% RSLogix 500 project LVD190506v3_Bot.RSS, saved by version 11.00.00.00 %
PROJECT "LINCEBOT"    % processor: MicroLogix 1400 %

PROGRAM FILES
  LAD 2 "MAIN"  40 rungs  % Main Program Routine %
  LAD 4 "PACKAGER"  27 rungs  % normal %
  LAD 5 "NO PACKAGE"  7 rungs
  LAD 6 "TIMING"  11 rungs  % normal %
  LAD 8 "LOOP TIME"  6 rungs
  LAD 10 "AIR PRESUR"  2 rungs
  LAD 12 "ENABLES"  13 rungs
  LAD 14 "SPEED OUT"  10 rungs
  LAD 16 "TOTALCOUNT"  4 rungs
  LAD 18 "TESTTRIG1"  4 rungs
  LAD 24 "SKIPPED"  5 rungs
  LAD 70 "ALIGNFAILS"  4 rungs  % normal %
  LAD 80 "HSC BOT"  5 rungs
  LAD 100 "1 MS STI"  19 rungs  % high speed %
  LAD 102 "SPEED BOT"  8 rungs  % high speed %
  LAD 104 "P BOT"  9 rungs  % high speed %
  LAD 110 "SHIFT BOT"  10 rungs
  LAD 120 "BOTOPTIC"  3 rungs
  LAD 121 "BOTOPTMES"  8 rungs
  LAD 129   1 rungs  % used for analysis %
  LAD 130 "INS1"  21 rungs
  LAD 131 "INS1RESULT"  7 rungs
  LAD 132 "INS1PASS"  3 rungs
  LAD 133 "INS1FAIL"  3 rungs
  LAD 134 "INS1ACQ"  8 rungs
  LAD 135 "Q1TIMETEST"  5 rungs
  LAD 136 "INS1TRIG"  5 rungs
  LAD 137 "FIFO1SET"  9 rungs
  LAD 138 "FIFO1GET"  8 rungs
  LAD 139 "INSDATA1"  3 rungs  % used for analysis %
  LAD 140 "TESTFAULT1"  9 rungs
  LAD 141 "INS1FIX1"  6 rungs
  LAD 142 "INS1FIX2"  3 rungs
  LAD 143 "HS TRIG1"  5 rungs
  LAD 200 "XFEROUT"  3 rungs
  LAD 201 "XFER GOOD"  5 rungs
  LAD 202 "XFER NG"  5 rungs
  LAD 222 "RATE1"  9 rungs
  LAD 223 "RATE2"  6 rungs
  LAD 224 "RESET RATE"  6 rungs
  LAD 122, 123, 124, 125, 126, 127, 128, 144, 145: only END

DATA FILES
  O0 OUTPUT  11 elements
  I1 INPUT  11 elements
  S2 STATUS  66 elements
  B3 BINARY  14 elements
  T4 TIMER  40 elements
  C5 COUNTER  1 elements
  R6 CONTROL  20 elements
  N7 INTEGER  200 elements
  F8 FLOAT  100 elements
  B9 TOP BS DAT  256 elements
  B10 OLD_COM  1 elements
  B11 BOT BS DAT  256 elements
  B12 HMI_BINARY  22 elements  % general use with hmi to avoid additional reads %
  L13  COUNTS  256 elements
  F14 HMI_FLOATS  100 elements
  N15 HMI_INTS  100 elements
  L16 HMI_LONGS  100 elements
  B17 SIDE DATA  128 elements
  B18 TOP DATA  128 elements
  L19 INS1TIME  10 elements
  L20 INS1POS  10 elements
  L21 INS5TIME  10 elements
  L22 INS5POS  10 elements
  L23 NEW READ  100 elements
  L24 NEW WRITE  100 elements
  L25 INS6TIME  10 elements
  L26 INS6POS  10 elements
  L27 RATETIMES  50 elements
  L28 INS1TIME  50 elements
  L29 INS1POS  50 elements
  L42   52 elements
  B181 BLANK  256 elements  % used to wipe bs files %
  F182 TEST FLOAT  50 elements
  L183 TEST LONG  50 elements
  N184 TEST INTS  50 elements
  B185 TEST BITS  50 elements
  N186 HMI INTS  50 elements
  L187 HMI LONG  50 elements
  F188 HMI FLOAT  50 elements
  B189 HMI BITS  50 elements
  L190 COUNTS  50 elements
  B191 ERROR BITS  10 elements
  L192 SPD OFFSET  50 elements
  F193 SPD OFFSET  50 elements
  B194 BOT GOOD  128 elements
  B195 BOT NG  128 elements
  B196 CTRL BITS  50 elements
  N197 CTRL INTS  50 elements
  B198 TRK BITS  50 elements
  L199 TRK LONG  50 elements
  N200 TRK INTS  50 elements
  L201 INS LONG  50 elements
  B202 INS BITS  50 elements
  N203 INS INTS  50 elements
  L204 CTRL LONG  50 elements
  F205 CTRL FLTS  50 elements

LADDER 2 "MAIN"    % Main Program Routine %
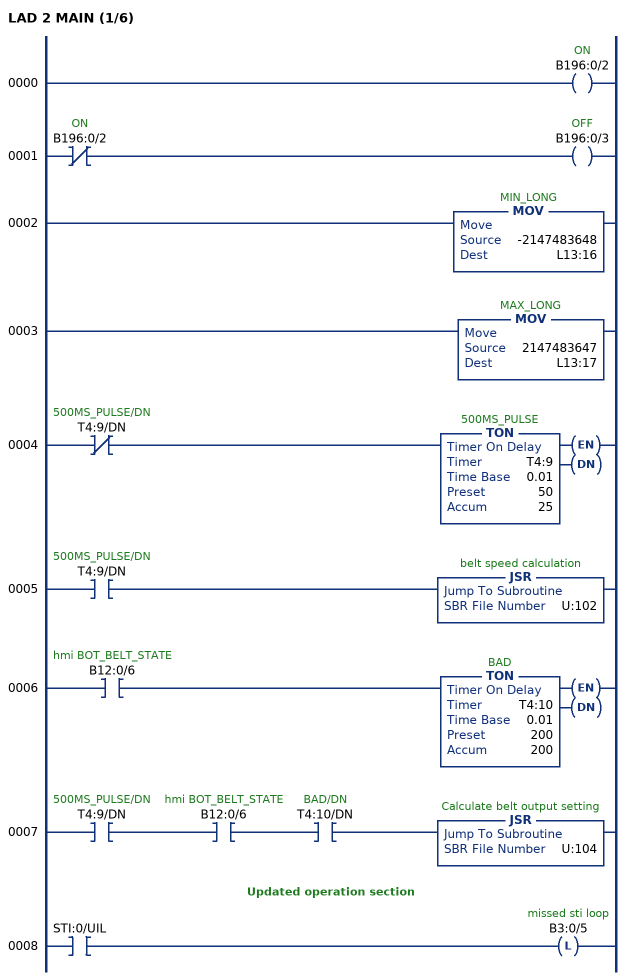
% Rung: 0 %
SOR OTE B196:0/2 EOR
%   B196:0/2  ON %
% Rung: 1 %
SOR XIO B196:0/2 OTE B196:0/3 EOR
%   B196:0/2  ON %
%   B196:0/3  OFF %
% Rung: 2 %
SOR MOV -2147483648 L13:16 EOR
%   L13:16  MIN_LONG %
% Rung: 3 %
SOR MOV 2147483647 L13:17 EOR
%   L13:17  MAX_LONG %
% Rung: 4 %
SOR XIO T4:9/DN TON T4:9 0.01 50 25 EOR
%   T4:9  500MS_PULSE %
% Rung: 5 %
SOR XIC T4:9/DN JSR U:102 EOR
%   T4:9  500MS_PULSE %
%   U:102  "belt speed calculation" %
% Rung: 6 %
SOR XIC B12:0/6 TON T4:10 0.01 200 200 EOR
%   B12:0/6  BOT_BELT_STATE  "hmi" %
%   T4:10  BAD %
% Rung: 7 %
SOR XIC T4:9/DN XIC B12:0/6 XIC T4:10/DN JSR U:104 EOR
%   T4:9  500MS_PULSE %
%   B12:0/6  BOT_BELT_STATE  "hmi" %
%   T4:10  BAD %
%   U:104  "Calculate belt output setting" %
% Rung: 8 %
% TITLE: Updated operation section %
SOR XIC STI:0/UIL OTL B3:0/5 EOR
%   B3:0/5  "missed sti loop" %

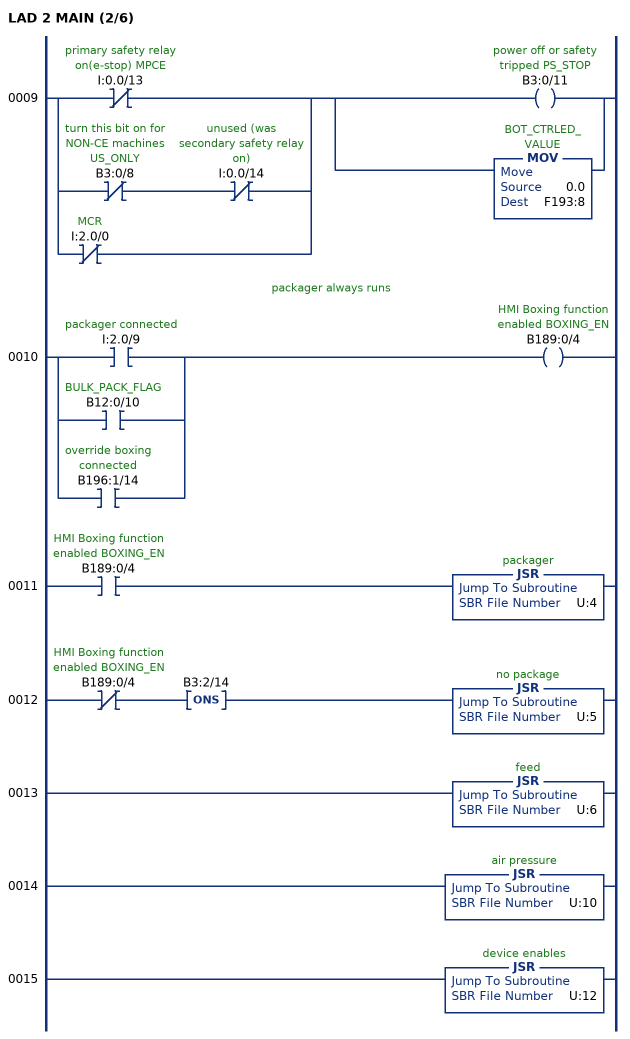
% Rung: 9 %
SOR BST XIO I:0.0/13 NXB XIO B3:0/8 XIO I:0.0/14 NXB XIO I:2.0/0 BND BST OTE B3:0/11 NXB MOV 0.0 F193:8 BND EOR
%   I:0.0/13  MPCE  "primary safety relay on(e-stop)" %
%   B3:0/8  US_ONLY  "turn this bit on for NON-CE machines" %
%   I:0.0/14  "unused (was secondary safety relay on)" %
%   I:2.0/0  MCR %
%   B3:0/11  PS_STOP  "power off or safety tripped" %
%   F193:8  BOT_CTRLED_VALUE %
% Rung: 10 %
% packager always runs %
SOR BST XIC I:2.0/9 NXB XIC B12:0/10 NXB XIC B196:1/14 BND OTE B189:0/4 EOR
%   I:2.0/9  "packager connected" %
%   B12:0/10  BULK_PACK_FLAG %
%   B196:1/14  "override boxing connected" %
%   B189:0/4  BOXING_EN  "HMI Boxing function enabled" %
% Rung: 11 %
SOR XIC B189:0/4 JSR U:4 EOR
%   B189:0/4  BOXING_EN  "HMI Boxing function enabled" %
%   U:4  "packager" %
% Rung: 12 %
SOR XIO B189:0/4 ONS B3:2/14 JSR U:5 EOR
%   B189:0/4  BOXING_EN  "HMI Boxing function enabled" %
%   U:5  "no package" %
% Rung: 13 %
SOR JSR U:6 EOR
%   U:6  "feed" %
% Rung: 14 %
SOR JSR U:10 EOR
%   U:10  "air pressure" %
% Rung: 15 %
SOR JSR U:12 EOR
%   U:12  "device enables" %

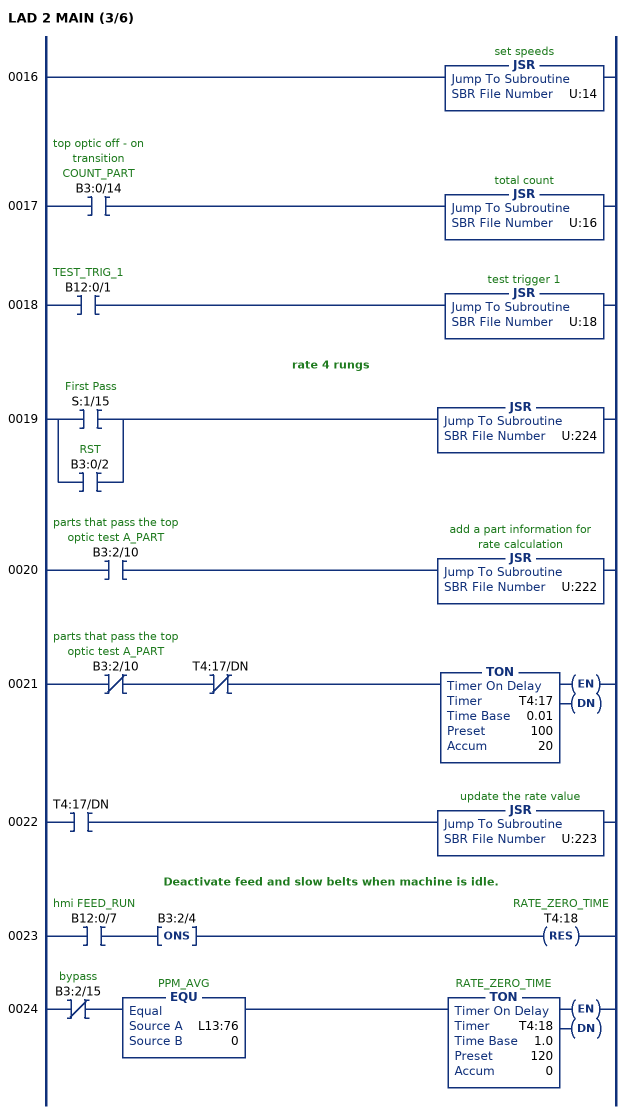
% Rung: 16 %
SOR JSR U:14 EOR
%   U:14  "set speeds" %
% Rung: 17 %
SOR XIC B3:0/14 JSR U:16 EOR
%   B3:0/14  COUNT_PART  "top optic off - on transition" %
%   U:16  "total count" %
% Rung: 18 %
SOR XIC B12:0/1 JSR U:18 EOR
%   B12:0/1  TEST_TRIG_1 %
%   U:18  "test trigger 1" %
% Rung: 19 %
% TITLE: rate 4 rungs %
SOR BST XIC S:1/15 NXB XIC B3:0/2 BND JSR U:224 EOR
%   S:1/15  "First Pass" %
%   B3:0/2  RST %
% Rung: 20 %
SOR XIC B3:2/10 JSR U:222 EOR
%   B3:2/10  A_PART  "parts that pass the top optic test" %
%   U:222  "add a part information for rate calculation" %
% Rung: 21 %
SOR XIO B3:2/10 XIO T4:17/DN TON T4:17 0.01 100 20 EOR
%   B3:2/10  A_PART  "parts that pass the top optic test" %
% Rung: 22 %
SOR XIC T4:17/DN JSR U:223 EOR
%   U:223  "update the rate value" %
% Rung: 23 %
% TITLE: Deactivate feed and slow belts when machine is idle. %
SOR XIC B12:0/7 ONS B3:2/4 RES T4:18 EOR
%   B12:0/7  FEED_RUN  "hmi" %
%   T4:18  RATE_ZERO_TIME %
% Rung: 24 %
SOR XIO B3:2/15 EQU L13:76 0 TON T4:18 1.0 120 0 EOR
%   B3:2/15  "bypass" %
%   L13:76  PPM_AVG %
%   T4:18  RATE_ZERO_TIME %

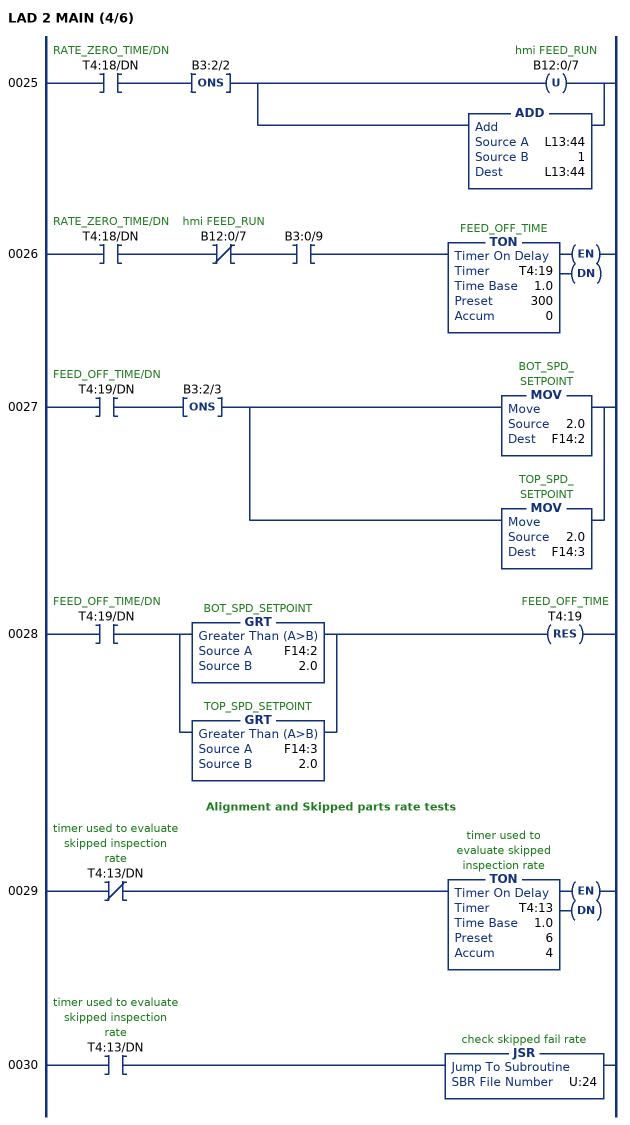
% Rung: 25 %
SOR XIC T4:18/DN ONS B3:2/2 BST OTU B12:0/7 NXB ADD L13:44 1 L13:44 BND EOR
%   T4:18  RATE_ZERO_TIME %
%   B12:0/7  FEED_RUN  "hmi" %
% Rung: 26 %
SOR XIC T4:18/DN XIO B12:0/7 XIC B3:0/9 TON T4:19 1.0 300 0 EOR
%   T4:18  RATE_ZERO_TIME %
%   B12:0/7  FEED_RUN  "hmi" %
%   T4:19  FEED_OFF_TIME %
% Rung: 27 %
SOR XIC T4:19/DN ONS B3:2/3 BST MOV 2.0 F14:2 NXB MOV 2.0 F14:3 BND EOR
%   T4:19  FEED_OFF_TIME %
%   F14:2  BOT_SPD_SETPOINT %
%   F14:3  TOP_SPD_SETPOINT %
% Rung: 28 %
SOR XIC T4:19/DN BST GRT F14:2 2.0 NXB GRT F14:3 2.0 BND RES T4:19 EOR
%   T4:19  FEED_OFF_TIME %
%   F14:2  BOT_SPD_SETPOINT %
%   F14:3  TOP_SPD_SETPOINT %
% Rung: 29 %
% TITLE: Alignment and Skipped parts rate tests %
SOR XIO T4:13/DN TON T4:13 1.0 6 4 EOR
%   T4:13  "timer used to evaluate skipped inspection rate" %
% Rung: 30 %
SOR XIC T4:13/DN JSR U:24 EOR
%   T4:13  "timer used to evaluate skipped inspection rate" %
%   U:24  "check skipped fail rate" %

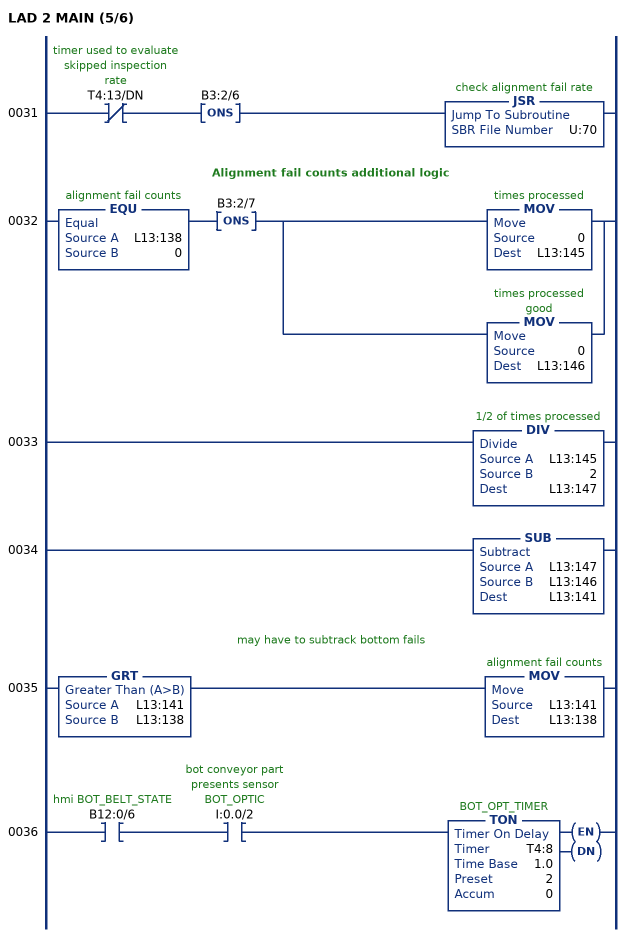
% Rung: 31 %
SOR XIO T4:13/DN ONS B3:2/6 JSR U:70 EOR
%   T4:13  "timer used to evaluate skipped inspection rate" %
%   U:70  "check alignment fail rate" %
% Rung: 32 %
% TITLE: Alignment fail counts additional logic %
SOR EQU L13:138 0 ONS B3:2/7 BST MOV 0 L13:145 NXB MOV 0 L13:146 BND EOR
%   L13:138  "alignment fail counts" %
%   L13:145  "times processed" %
%   L13:146  "times processed good" %
% Rung: 33 %
SOR DIV L13:145 2 L13:147 EOR
%   L13:145  "times processed" %
%   L13:147  "1/2 of times processed" %
% Rung: 34 %
SOR SUB L13:147 L13:146 L13:141 EOR
%   L13:147  "1/2 of times processed" %
%   L13:146  "times processed good" %
% Rung: 35 %
% may have to subtrack bottom fails %
SOR GRT L13:141 L13:138 MOV L13:141 L13:138 EOR
%   L13:138  "alignment fail counts" %
% Rung: 36 %
SOR XIC B12:0/6 XIC I:0.0/2 TON T4:8 1.0 2 0 EOR
%   B12:0/6  BOT_BELT_STATE  "hmi" %
%   I:0.0/2  BOT_OPTIC  "bot conveyor part presents sensor" %
%   T4:8  BOT_OPT_TIMER %

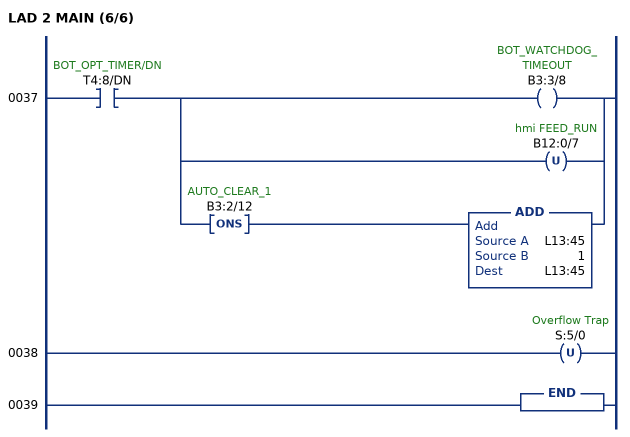
% Rung: 37 %
SOR XIC T4:8/DN BST OTE B3:3/8 NXB OTU B12:0/7 NXB ONS B3:2/12 ADD L13:45 1 L13:45 BND EOR
%   T4:8  BOT_OPT_TIMER %
%   B3:3/8  BOT_WATCHDOG_TIMEOUT %
%   B12:0/7  FEED_RUN  "hmi" %
%   B3:2/12  AUTO_CLEAR_1 %
% Rung: 38 %
SOR OTU S:5/0 EOR
%   S:5/0  "Overflow Trap" %
% Rung: 39 %
SOR END EOR

LADDER 4 "PACKAGER"    % normal %
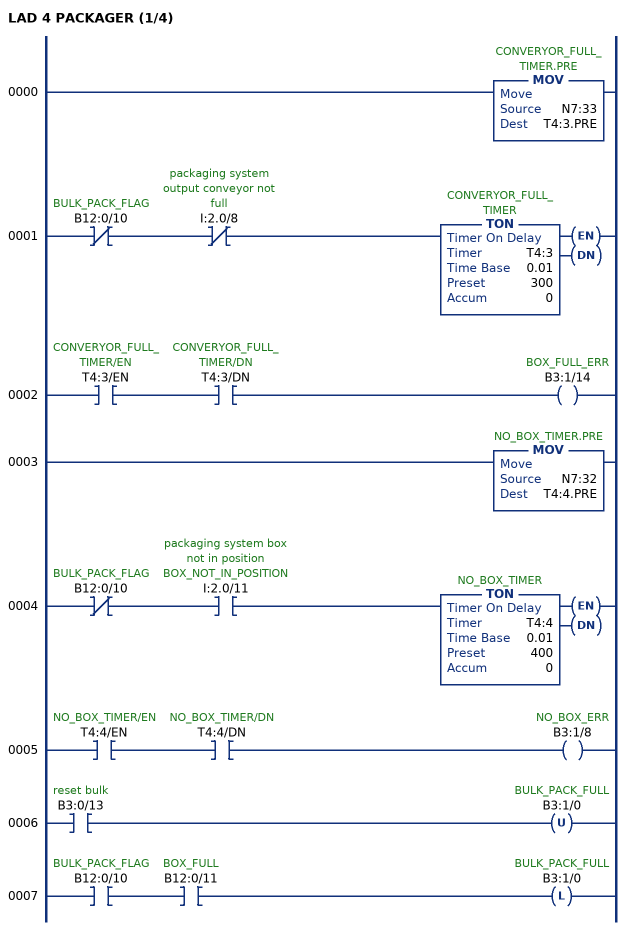
% Rung: 0 %
SOR MOV N7:33 T4:3.PRE EOR
%   T4:3  CONVERYOR_FULL_TIMER %
% Rung: 1 %
SOR XIO B12:0/10 XIO I:2.0/8 TON T4:3 0.01 300 0 EOR
%   B12:0/10  BULK_PACK_FLAG %
%   I:2.0/8  "packaging system output conveyor not full" %
%   T4:3  CONVERYOR_FULL_TIMER %
% Rung: 2 %
SOR XIC T4:3/EN XIC T4:3/DN OTE B3:1/14 EOR
%   T4:3  CONVERYOR_FULL_TIMER %
%   B3:1/14  BOX_FULL_ERR %
% Rung: 3 %
SOR MOV N7:32 T4:4.PRE EOR
%   T4:4  NO_BOX_TIMER %
% Rung: 4 %
SOR XIO B12:0/10 XIC I:2.0/11 TON T4:4 0.01 400 0 EOR
%   B12:0/10  BULK_PACK_FLAG %
%   I:2.0/11  BOX_NOT_IN_POSITION  "packaging system box not in position" %
%   T4:4  NO_BOX_TIMER %
% Rung: 5 %
SOR XIC T4:4/EN XIC T4:4/DN OTE B3:1/8 EOR
%   T4:4  NO_BOX_TIMER %
%   B3:1/8  NO_BOX_ERR %
% Rung: 6 %
SOR XIC B3:0/13 OTU B3:1/0 EOR
%   B3:0/13  "reset bulk" %
%   B3:1/0  BULK_PACK_FULL %
% Rung: 7 %
SOR XIC B12:0/10 XIC B12:0/11 OTL B3:1/0 EOR
%   B12:0/10  BULK_PACK_FLAG %
%   B12:0/11  BOX_FULL %
%   B3:1/0  BULK_PACK_FULL %

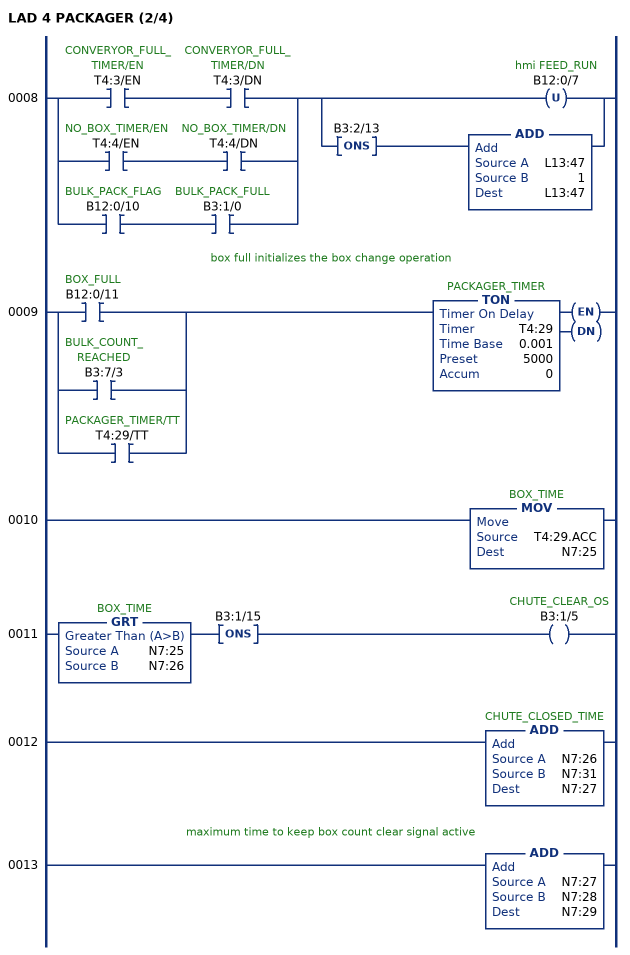
% Rung: 8 %
SOR BST XIC T4:3/EN XIC T4:3/DN NXB XIC T4:4/EN XIC T4:4/DN NXB XIC B12:0/10 XIC B3:1/0 BND BST OTU B12:0/7 NXB ONS B3:2/13 ADD L13:47 1 L13:47 BND EOR
%   T4:3  CONVERYOR_FULL_TIMER %
%   T4:4  NO_BOX_TIMER %
%   B12:0/10  BULK_PACK_FLAG %
%   B3:1/0  BULK_PACK_FULL %
%   B12:0/7  FEED_RUN  "hmi" %
% Rung: 9 %
% box full initializes the box change operation %
SOR BST XIC B12:0/11 NXB XIC B3:7/3 NXB XIC T4:29/TT BND TON T4:29 0.001 5000 0 EOR
%   B12:0/11  BOX_FULL %
%   B3:7/3  BULK_COUNT_REACHED %
%   T4:29  PACKAGER_TIMER %
% Rung: 10 %
SOR MOV T4:29.ACC N7:25 EOR
%   T4:29  PACKAGER_TIMER %
%   N7:25  BOX_TIME %
% Rung: 11 %
SOR GRT N7:25 N7:26 ONS B3:1/15 OTE B3:1/5 EOR
%   N7:25  BOX_TIME %
%   N7:26  CHUTE_CLEAR_TIME %
%   B3:1/5  CHUTE_CLEAR_OS %
% Rung: 12 %
SOR ADD N7:26 N7:31 N7:27 EOR
%   N7:26  CHUTE_CLEAR_TIME %
%   N7:27  CHUTE_CLOSED_TIME %
% Rung: 13 %
% maximum time to keep box count clear signal active %
SOR ADD N7:27 N7:28 N7:29 EOR
%   N7:27  CHUTE_CLOSED_TIME %

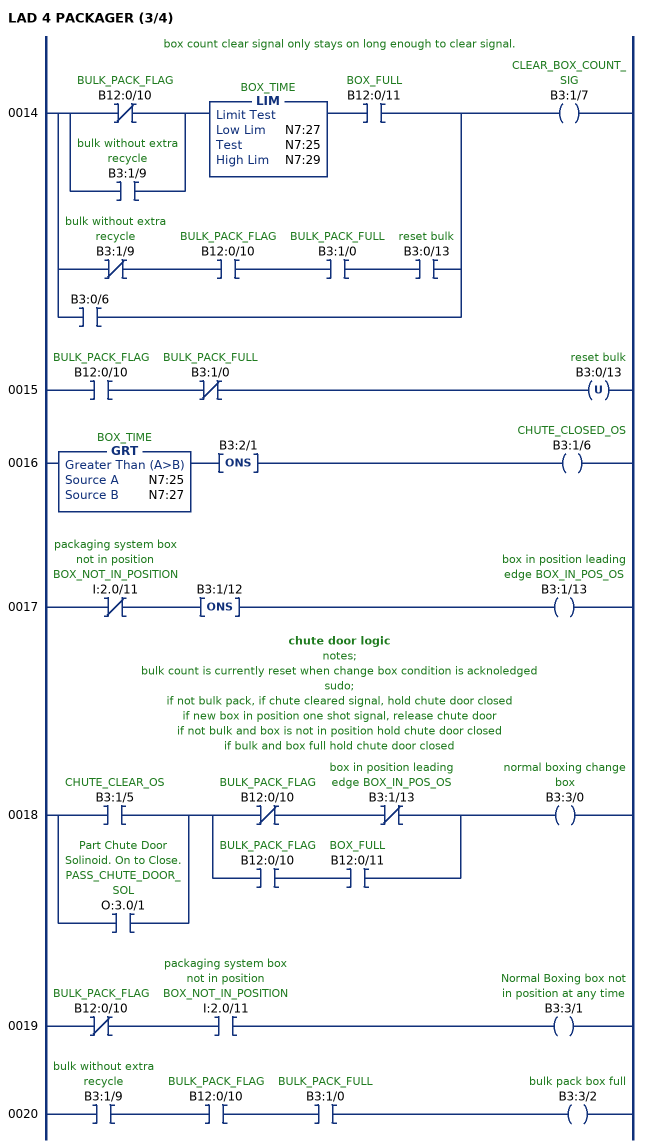
% Rung: 14 %
% box count clear signal only stays on long enough to clear signal. %
SOR BST BST XIO B12:0/10 NXB XIC B3:1/9 BND LIM N7:27 N7:25 N7:29 XIC B12:0/11 NXB XIO B3:1/9 XIC B12:0/10 XIC B3:1/0 XIC B3:0/13 NXB XIC B3:0/6 BND OTE B3:1/7 EOR
%   B12:0/10  BULK_PACK_FLAG %
%   B3:1/9  "bulk without extra recycle" %
%   N7:27  CHUTE_CLOSED_TIME %
%   N7:25  BOX_TIME %
%   B12:0/11  BOX_FULL %
%   B3:1/0  BULK_PACK_FULL %
%   B3:0/13  "reset bulk" %
%   B3:1/7  CLEAR_BOX_COUNT_SIG %
% Rung: 15 %
SOR XIC B12:0/10 XIO B3:1/0 OTU B3:0/13 EOR
%   B12:0/10  BULK_PACK_FLAG %
%   B3:1/0  BULK_PACK_FULL %
%   B3:0/13  "reset bulk" %
% Rung: 16 %
SOR GRT N7:25 N7:27 ONS B3:2/1 OTE B3:1/6 EOR
%   N7:25  BOX_TIME %
%   N7:27  CHUTE_CLOSED_TIME %
%   B3:1/6  CHUTE_CLOSED_OS %
% Rung: 17 %
SOR XIO I:2.0/11 ONS B3:1/12 OTE B3:1/13 EOR
%   I:2.0/11  BOX_NOT_IN_POSITION  "packaging system box not in position" %
%   B3:1/13  BOX_IN_POS_OS  "box in position leading edge" %
% Rung: 18 %
% TITLE: chute door logic %
% notes;
% bulk count is currently reset when change box condition is acknoledged
% 
% sudo;
% if not bulk pack, if chute cleared signal, hold chute door closed
%           if new box in position one shot signal, release chute door
% if not bulk and box is not in position hold chute door closed
% if bulk and box full hold chute door closed %
SOR BST XIC B3:1/5 NXB XIC O:3.0/1 BND BST XIO B12:0/10 XIO B3:1/13 NXB XIC B12:0/10 XIC B12:0/11 BND OTE B3:3/0 EOR
%   B3:1/5  CHUTE_CLEAR_OS %
%   O:3.0/1  PASS_CHUTE_DOOR_SOL  "Part Chute Door Solinoid. On to Close." %
%   B12:0/10  BULK_PACK_FLAG %
%   B3:1/13  BOX_IN_POS_OS  "box in position leading edge" %
%   B12:0/11  BOX_FULL %
%   B3:3/0  "normal boxing change box" %
% Rung: 19 %
SOR XIO B12:0/10 XIC I:2.0/11 OTE B3:3/1 EOR
%   B12:0/10  BULK_PACK_FLAG %
%   I:2.0/11  BOX_NOT_IN_POSITION  "packaging system box not in position" %
%   B3:3/1  "Normal Boxing box not in position at any time" %
% Rung: 20 %
SOR XIC B3:1/9 XIC B12:0/10 XIC B3:1/0 OTE B3:3/2 EOR
%   B3:1/9  "bulk without extra recycle" %
%   B12:0/10  BULK_PACK_FLAG %
%   B3:1/0  BULK_PACK_FULL %
%   B3:3/2  "bulk pack box full" %

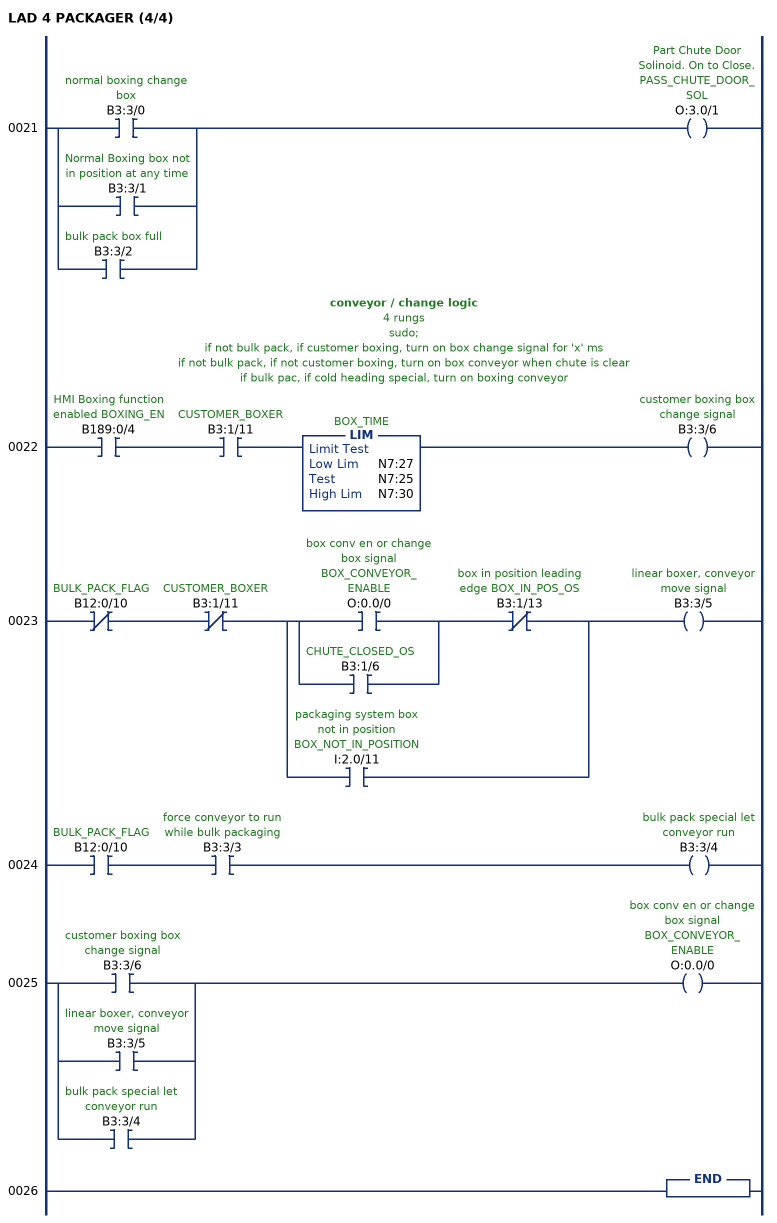
% Rung: 21 %
SOR BST XIC B3:3/0 NXB XIC B3:3/1 NXB XIC B3:3/2 BND OTE O:3.0/1 EOR
%   B3:3/0  "normal boxing change box" %
%   B3:3/1  "Normal Boxing box not in position at any time" %
%   B3:3/2  "bulk pack box full" %
%   O:3.0/1  PASS_CHUTE_DOOR_SOL  "Part Chute Door Solinoid. On to Close." %
% Rung: 22 %
% TITLE: conveyor / change logic %
% 4 rungs
% sudo;
% if not bulk pack, if customer boxing, turn on box change signal for 'x' ms
% if not bulk pack, if not customer boxing, turn on box conveyor when chute is clear
% if bulk pac, if cold heading special, turn on boxing conveyor %
SOR XIC B189:0/4 XIC B3:1/11 LIM N7:27 N7:25 N7:30 OTE B3:3/6 EOR
%   B189:0/4  BOXING_EN  "HMI Boxing function enabled" %
%   B3:1/11  CUSTOMER_BOXER %
%   N7:27  CHUTE_CLOSED_TIME %
%   N7:25  BOX_TIME %
%   N7:30  END_OF_CHANGE_SIG %
%   B3:3/6  "customer boxing box change signal" %
% Rung: 23 %
SOR XIO B12:0/10 XIO B3:1/11 BST BST XIC O:0.0/0 NXB XIC B3:1/6 BND XIO B3:1/13 NXB XIC I:2.0/11 BND OTE B3:3/5 EOR
%   B12:0/10  BULK_PACK_FLAG %
%   B3:1/11  CUSTOMER_BOXER %
%   O:0.0/0  BOX_CONVEYOR_ENABLE  "box conv en or change box signal" %
%   B3:1/6  CHUTE_CLOSED_OS %
%   B3:1/13  BOX_IN_POS_OS  "box in position leading edge" %
%   I:2.0/11  BOX_NOT_IN_POSITION  "packaging system box not in position" %
%   B3:3/5  "linear boxer, conveyor move signal" %
% Rung: 24 %
SOR XIC B12:0/10 XIC B3:3/3 OTE B3:3/4 EOR
%   B12:0/10  BULK_PACK_FLAG %
%   B3:3/3  "force conveyor to run while bulk packaging" %
%   B3:3/4  "bulk pack special let conveyor run" %
% Rung: 25 %
SOR BST XIC B3:3/6 NXB XIC B3:3/5 NXB XIC B3:3/4 BND OTE O:0.0/0 EOR
%   B3:3/6  "customer boxing box change signal" %
%   B3:3/5  "linear boxer, conveyor move signal" %
%   B3:3/4  "bulk pack special let conveyor run" %
%   O:0.0/0  BOX_CONVEYOR_ENABLE  "box conv en or change box signal" %
% Rung: 26 %
SOR END EOR

LADDER 5 "NO PACKAGE"
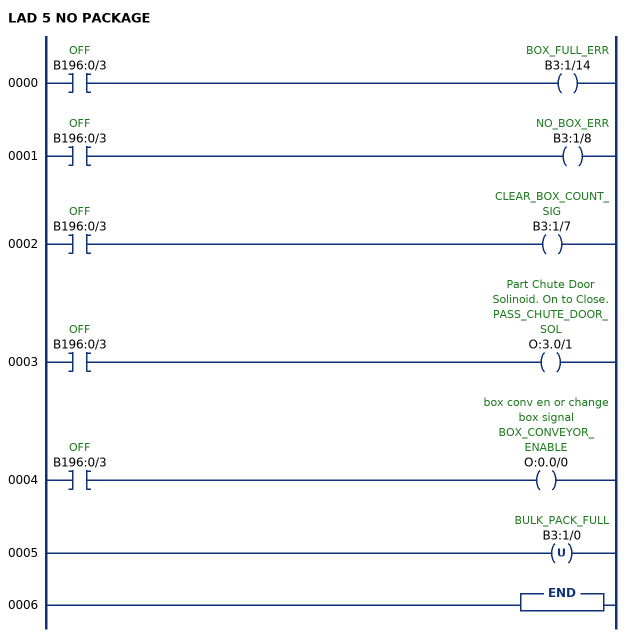
% Rung: 0 %
SOR XIC B196:0/3 OTE B3:1/14 EOR
%   B196:0/3  OFF %
%   B3:1/14  BOX_FULL_ERR %
% Rung: 1 %
SOR XIC B196:0/3 OTE B3:1/8 EOR
%   B196:0/3  OFF %
%   B3:1/8  NO_BOX_ERR %
% Rung: 2 %
SOR XIC B196:0/3 OTE B3:1/7 EOR
%   B196:0/3  OFF %
%   B3:1/7  CLEAR_BOX_COUNT_SIG %
% Rung: 3 %
SOR XIC B196:0/3 OTE O:3.0/1 EOR
%   B196:0/3  OFF %
%   O:3.0/1  PASS_CHUTE_DOOR_SOL  "Part Chute Door Solinoid. On to Close." %
% Rung: 4 %
SOR XIC B196:0/3 OTE O:0.0/0 EOR
%   B196:0/3  OFF %
%   O:0.0/0  BOX_CONVEYOR_ENABLE  "box conv en or change box signal" %
% Rung: 5 %
SOR OTU B3:1/0 EOR
%   B3:1/0  BULK_PACK_FULL %
% Rung: 6 %
SOR END EOR

LADDER 6 "TIMING"    % normal %
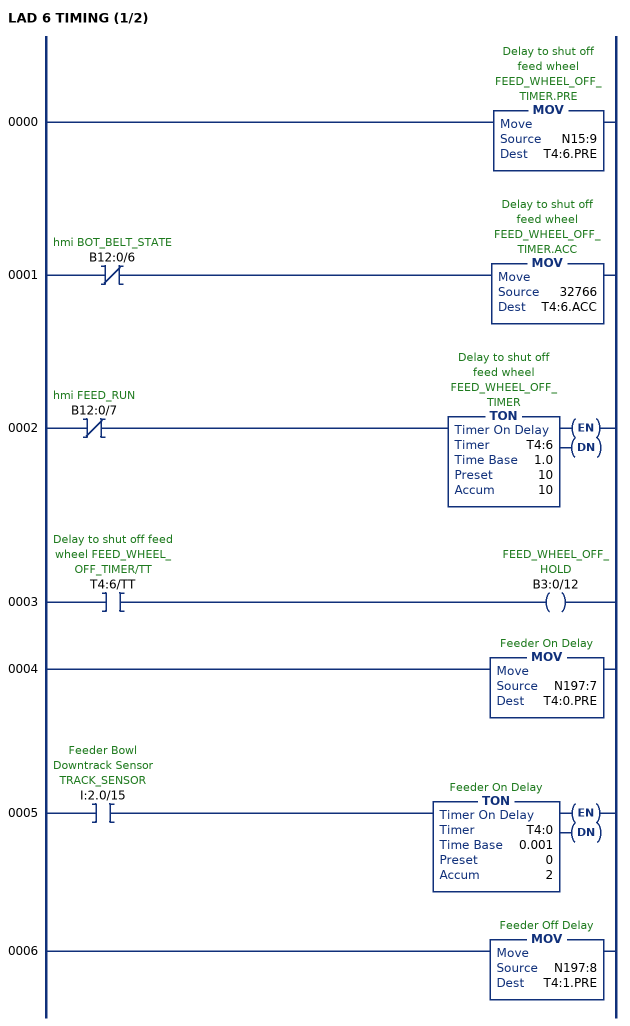
% Rung: 0 %
SOR MOV N15:9 T4:6.PRE EOR
%   N15:9  FEED_WHEEL_STOP_TIME %
%   T4:6  FEED_WHEEL_OFF_TIMER  "Delay to shut off feed wheel" %
% Rung: 1 %
SOR XIO B12:0/6 MOV 32766 T4:6.ACC EOR
%   B12:0/6  BOT_BELT_STATE  "hmi" %
%   T4:6  FEED_WHEEL_OFF_TIMER  "Delay to shut off feed wheel" %
% Rung: 2 %
SOR XIO B12:0/7 TON T4:6 1.0 10 10 EOR
%   B12:0/7  FEED_RUN  "hmi" %
%   T4:6  FEED_WHEEL_OFF_TIMER  "Delay to shut off feed wheel" %
% Rung: 3 %
SOR XIC T4:6/TT OTE B3:0/12 EOR
%   T4:6  FEED_WHEEL_OFF_TIMER  "Delay to shut off feed wheel" %
%   B3:0/12  FEED_WHEEL_OFF_HOLD %
% Rung: 4 %
SOR MOV N197:7 T4:0.PRE EOR
%   N197:7  "down track on delay" %
%   T4:0  "Feeder On Delay" %
% Rung: 5 %
SOR XIC I:2.0/15 TON T4:0 0.001 0 2 EOR
%   I:2.0/15  TRACK_SENSOR  "Feeder Bowl Downtrack Sensor" %
%   T4:0  "Feeder On Delay" %
% Rung: 6 %
SOR MOV N197:8 T4:1.PRE EOR
%   N197:8  "down track off delay" %
%   T4:1  "Feeder Off Delay" %

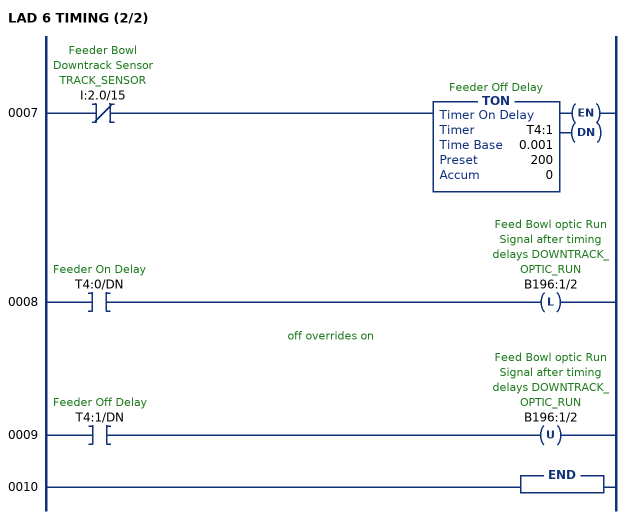
% Rung: 7 %
SOR XIO I:2.0/15 TON T4:1 0.001 200 0 EOR
%   I:2.0/15  TRACK_SENSOR  "Feeder Bowl Downtrack Sensor" %
%   T4:1  "Feeder Off Delay" %
% Rung: 8 %
SOR XIC T4:0/DN OTL B196:1/2 EOR
%   T4:0  "Feeder On Delay" %
%   B196:1/2  DOWNTRACK_OPTIC_RUN  "Feed Bowl optic Run Signal after timing delays" %
% Rung: 9 %
% off overrides on %
SOR XIC T4:1/DN OTU B196:1/2 EOR
%   T4:1  "Feeder Off Delay" %
%   B196:1/2  DOWNTRACK_OPTIC_RUN  "Feed Bowl optic Run Signal after timing delays" %
% Rung: 10 %
SOR END EOR

LADDER 8 "LOOP TIME"
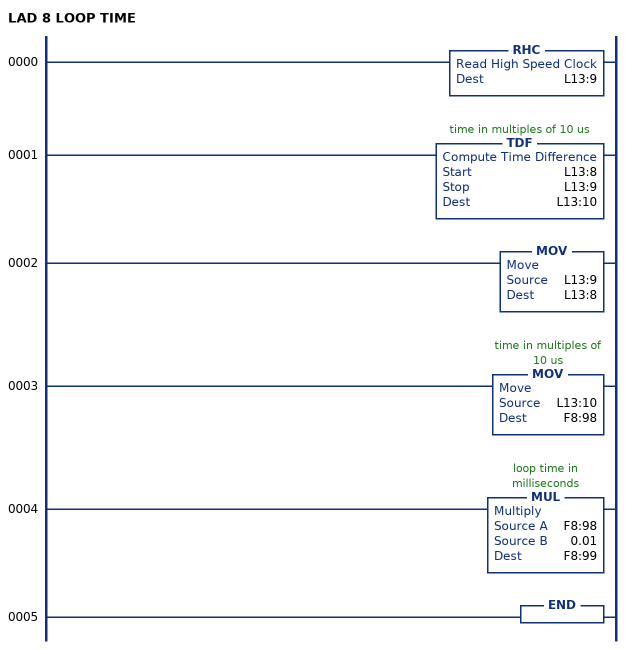
% Rung: 0 %
SOR RHC L13:9 EOR
% Rung: 1 %
SOR TDF L13:8 L13:9 L13:10 EOR
%   L13:10  "time in multiples of 10 us" %
% Rung: 2 %
SOR MOV L13:9 L13:8 EOR
% Rung: 3 %
SOR MOV L13:10 F8:98 EOR
%   L13:10  "time in multiples of 10 us" %
%   F8:98  "time in multiples of 10 us" %
% Rung: 4 %
SOR MUL F8:98 0.01 F8:99 EOR
%   F8:98  "time in multiples of 10 us" %
%   F8:99  "loop time in milliseconds" %
% Rung: 5 %
SOR END EOR

LADDER 10 "AIR PRESUR"
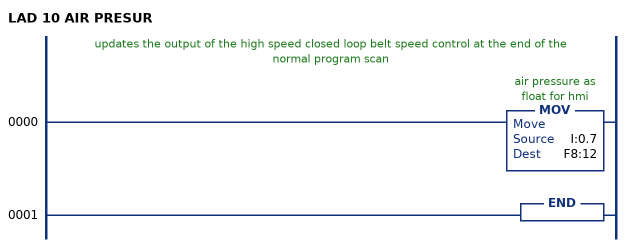
% Rung: 0 %
% updates the output of the high speed closed loop belt speed control at the end of the normal program scan %
SOR MOV I:0.7 F8:12 EOR
%   I:0.7  "Air Presure Sensor Input Signal" %
%   F8:12  "air pressure as float for hmi" %
% Rung: 1 %
SOR END EOR

LADDER 12 "ENABLES"
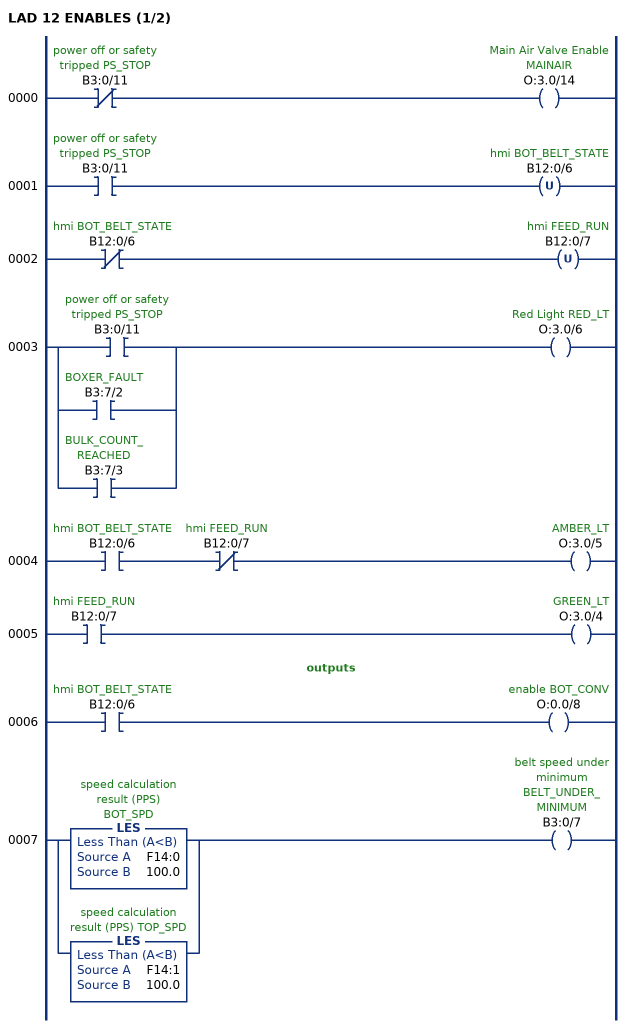
% Rung: 0 %
SOR XIO B3:0/11 OTE O:3.0/14 EOR
%   B3:0/11  PS_STOP  "power off or safety tripped" %
%   O:3.0/14  MAINAIR  "Main Air Valve Enable" %
% Rung: 1 %
SOR XIC B3:0/11 OTU B12:0/6 EOR
%   B3:0/11  PS_STOP  "power off or safety tripped" %
%   B12:0/6  BOT_BELT_STATE  "hmi" %
% Rung: 2 %
SOR XIO B12:0/6 OTU B12:0/7 EOR
%   B12:0/6  BOT_BELT_STATE  "hmi" %
%   B12:0/7  FEED_RUN  "hmi" %
% Rung: 3 %
SOR BST XIC B3:0/11 NXB XIC B3:7/2 NXB XIC B3:7/3 BND OTE O:3.0/6 EOR
%   B3:0/11  PS_STOP  "power off or safety tripped" %
%   B3:7/2  BOXER_FAULT %
%   B3:7/3  BULK_COUNT_REACHED %
%   O:3.0/6  RED_LT  "Red Light" %
% Rung: 4 %
SOR XIC B12:0/6 XIO B12:0/7 OTE O:3.0/5 EOR
%   B12:0/6  BOT_BELT_STATE  "hmi" %
%   B12:0/7  FEED_RUN  "hmi" %
%   O:3.0/5  AMBER_LT %
% Rung: 5 %
SOR XIC B12:0/7 OTE O:3.0/4 EOR
%   B12:0/7  FEED_RUN  "hmi" %
%   O:3.0/4  GREEN_LT %
% Rung: 6 %
% TITLE: outputs %
SOR XIC B12:0/6 OTE O:0.0/8 EOR
%   B12:0/6  BOT_BELT_STATE  "hmi" %
%   O:0.0/8  BOT_CONV  "enable" %
% Rung: 7 %
SOR BST LES F14:0 100.0 NXB LES F14:1 100.0 BND OTE B3:0/7 EOR
%   F14:0  BOT_SPD  "speed calculation result (PPS)" %
%   F14:1  TOP_SPD  "speed calculation result (PPS)" %
%   B3:0/7  BELT_UNDER_MINIMUM  "belt speed under minimum" %

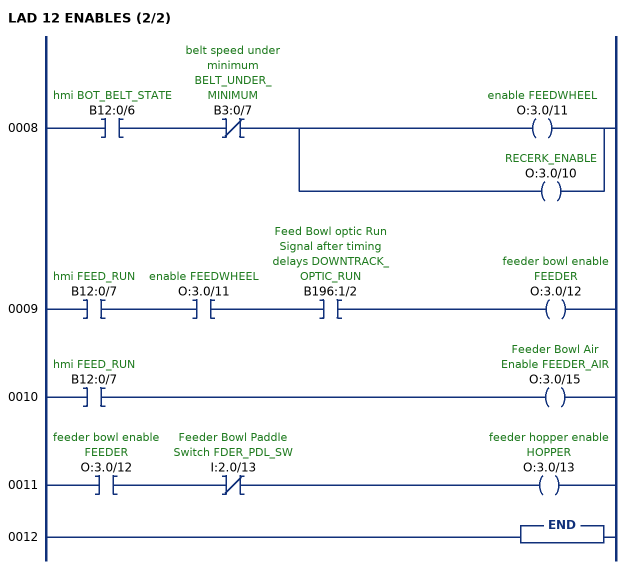
% Rung: 8 %
SOR XIC B12:0/6 XIO B3:0/7 BST OTE O:3.0/11 NXB OTE O:3.0/10 BND EOR
%   B12:0/6  BOT_BELT_STATE  "hmi" %
%   B3:0/7  BELT_UNDER_MINIMUM  "belt speed under minimum" %
%   O:3.0/11  FEEDWHEEL  "enable" %
%   O:3.0/10  RECERK_ENABLE %
% Rung: 9 %
SOR XIC B12:0/7 XIC O:3.0/11 XIC B196:1/2 OTE O:3.0/12 EOR
%   B12:0/7  FEED_RUN  "hmi" %
%   O:3.0/11  FEEDWHEEL  "enable" %
%   B196:1/2  DOWNTRACK_OPTIC_RUN  "Feed Bowl optic Run Signal after timing delays" %
%   O:3.0/12  FEEDER  "feeder bowl enable" %
% Rung: 10 %
SOR XIC B12:0/7 OTE O:3.0/15 EOR
%   B12:0/7  FEED_RUN  "hmi" %
%   O:3.0/15  FEEDER_AIR  "Feeder Bowl Air Enable" %
% Rung: 11 %
SOR XIC O:3.0/12 XIO I:2.0/13 OTE O:3.0/13 EOR
%   O:3.0/12  FEEDER  "feeder bowl enable" %
%   I:2.0/13  FDER_PDL_SW  "Feeder Bowl Paddle Switch" %
%   O:3.0/13  HOPPER  "feeder hopper enable" %
% Rung: 12 %
SOR END EOR

LADDER 14 "SPEED OUT"
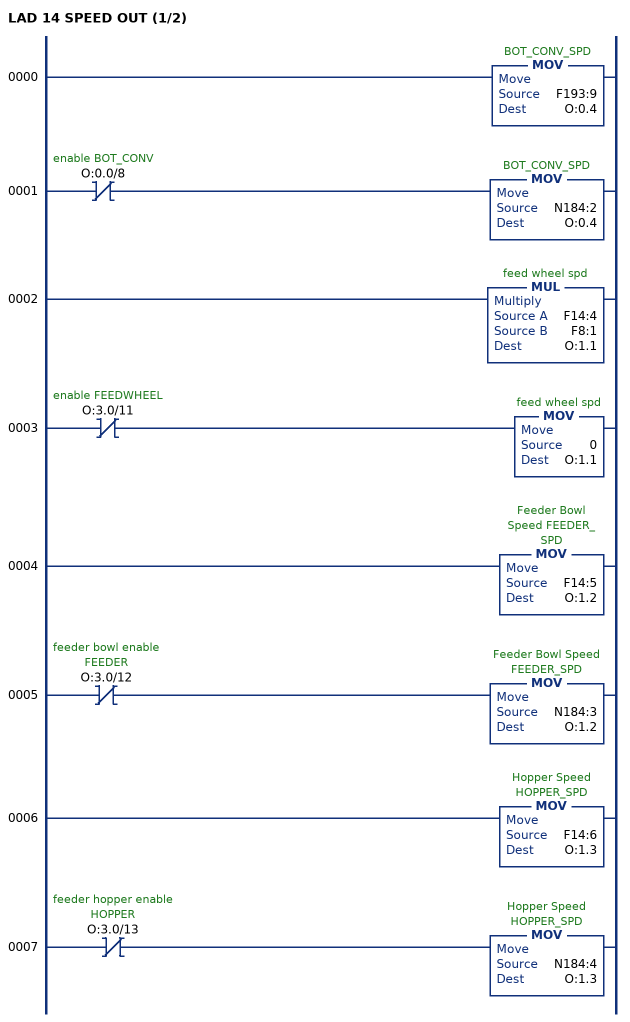
% Rung: 0 %
SOR MOV F193:9 O:0.4 EOR
%   F193:9  SCALED_BOT_VALUE %
%   O:0.4  BOT_CONV_SPD %
% Rung: 1 %
SOR XIO O:0.0/8 MOV N184:2 O:0.4 EOR
%   O:0.0/8  BOT_CONV  "enable" %
%   O:0.4  BOT_CONV_SPD %
% Rung: 2 %
SOR MUL F14:4 F8:1 O:1.1 EOR
%   F14:4  "feed wheel spd" %
%   O:1.1  "feed wheel spd" %
% Rung: 3 %
SOR XIO O:3.0/11 MOV 0 O:1.1 EOR
%   O:3.0/11  FEEDWHEEL  "enable" %
%   O:1.1  "feed wheel spd" %
% Rung: 4 %
SOR MOV F14:5 O:1.2 EOR
%   O:1.2  FEEDER_SPD  "Feeder Bowl Speed" %
% Rung: 5 %
SOR XIO O:3.0/12 MOV N184:3 O:1.2 EOR
%   O:3.0/12  FEEDER  "feeder bowl enable" %
%   O:1.2  FEEDER_SPD  "Feeder Bowl Speed" %
% Rung: 6 %
SOR MOV F14:6 O:1.3 EOR
%   O:1.3  HOPPER_SPD  "Hopper Speed" %
% Rung: 7 %
SOR XIO O:3.0/13 MOV N184:4 O:1.3 EOR
%   O:3.0/13  HOPPER  "feeder hopper enable" %
%   O:1.3  HOPPER_SPD  "Hopper Speed" %

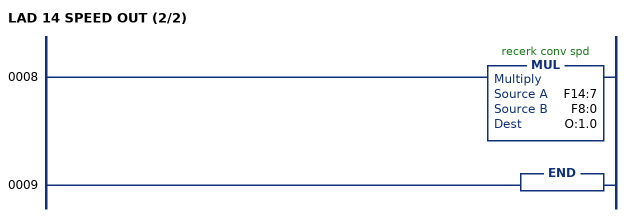
% Rung: 8 %
SOR MUL F14:7 F8:0 O:1.0 EOR
%   F14:7  "recerk speed setting" %
%   O:1.0  "recerk conv spd" %
% Rung: 9 %
SOR END EOR

LADDER 16 "TOTALCOUNT"
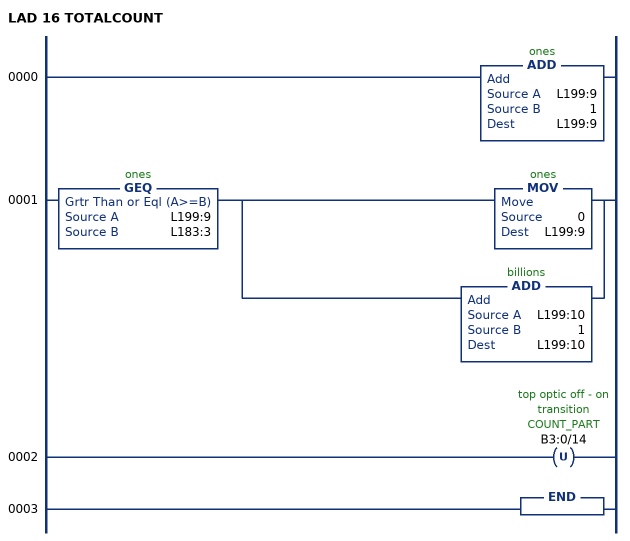
% Rung: 0 %
SOR ADD L199:9 1 L199:9 EOR
%   L199:9  "ones" %
% Rung: 1 %
SOR GEQ L199:9 L183:3 BST MOV 0 L199:9 NXB ADD L199:10 1 L199:10 BND EOR
%   L199:9  "ones" %
%   L183:3  "button state" %
%   L199:10  "billions" %
% Rung: 2 %
SOR OTU B3:0/14 EOR
%   B3:0/14  COUNT_PART  "top optic off - on transition" %
% Rung: 3 %
SOR END EOR

LADDER 18 "TESTTRIG1"
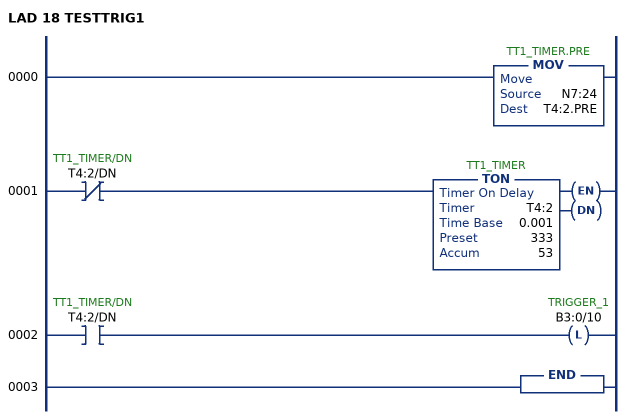
% Rung: 0 %
SOR MOV N7:24 T4:2.PRE EOR
%   T4:2  TT1_TIMER %
% Rung: 1 %
SOR XIO T4:2/DN TON T4:2 0.001 333 53 EOR
%   T4:2  TT1_TIMER %
% Rung: 2 %
SOR XIC T4:2/DN OTL B3:0/10 EOR
%   T4:2  TT1_TIMER %
%   B3:0/10  TRIGGER_1 %
% Rung: 3 %
SOR END EOR

LADDER 24 "SKIPPED"
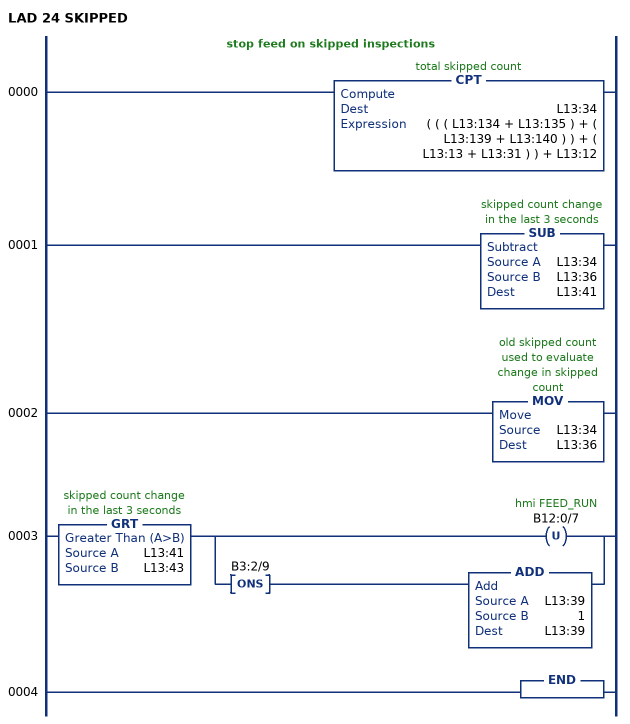
% Rung: 0 %
% TITLE: stop feed on skipped inspections %
SOR CPT L13:34 " ( ( ( L13:134 + L13:135 ) + ( L13:139 + L13:140 ) ) + ( L13:13 + L13:31 ) ) + L13:12 " EOR
%   L13:34  "total skipped count" %
%   L13:134  "too wide bottom" %
%   L13:135  "too close bottom" %
%   L13:139  "too close top count" %
%   L13:140  "too wide top count" %
%   L13:13  SKIP1  "skipped 1 count" %
%   L13:31  SKIP5  "skipped 5 count" %
%   L13:12  SKIP6  "skipped 6 count" %
% Rung: 1 %
SOR SUB L13:34 L13:36 L13:41 EOR
%   L13:34  "total skipped count" %
%   L13:36  "old skipped count used to evaluate change in skipped count" %
%   L13:41  "skipped count change in the last 3 seconds" %
% Rung: 2 %
SOR MOV L13:34 L13:36 EOR
%   L13:34  "total skipped count" %
%   L13:36  "old skipped count used to evaluate change in skipped count" %
% Rung: 3 %
SOR GRT L13:41 L13:43 BST OTU B12:0/7 NXB ONS B3:2/9 ADD L13:39 1 L13:39 BND EOR
%   L13:41  "skipped count change in the last 3 seconds" %
%   L13:43  "trigger count 1" %
%   B12:0/7  FEED_RUN  "hmi" %
% Rung: 4 %
SOR END EOR

LADDER 70 "ALIGNFAILS"    % normal %
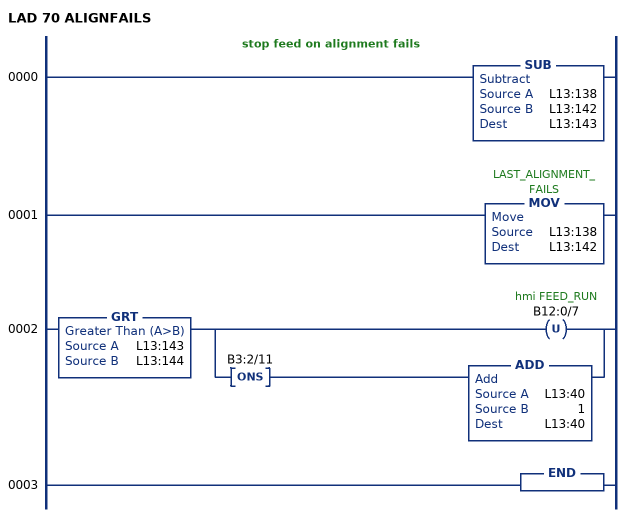
% Rung: 0 %
% TITLE: stop feed on alignment fails %
SOR SUB L13:138 L13:142 L13:143 EOR
%   L13:138  "alignment fail counts" %
%   L13:142  LAST_ALIGNMENT_FAILS %
% Rung: 1 %
SOR MOV L13:138 L13:142 EOR
%   L13:138  "alignment fail counts" %
%   L13:142  LAST_ALIGNMENT_FAILS %
% Rung: 2 %
SOR GRT L13:143 L13:144 BST OTU B12:0/7 NXB ONS B3:2/11 ADD L13:40 1 L13:40 BND EOR
%   B12:0/7  FEED_RUN  "hmi" %
% Rung: 3 %
SOR END EOR

LADDER 80 "HSC BOT"
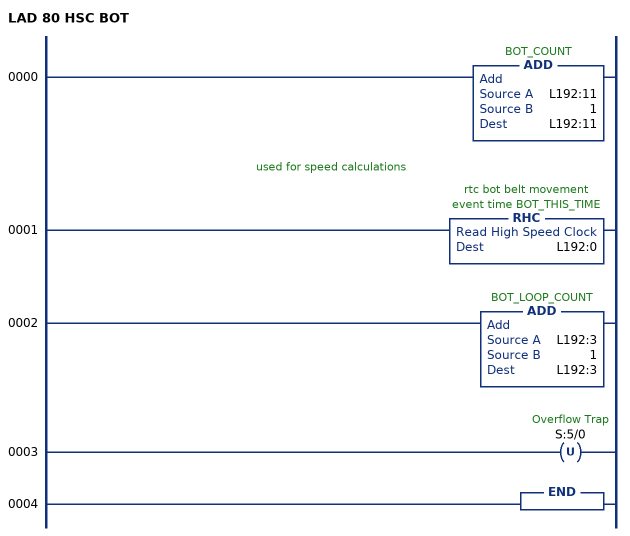
% Rung: 0 %
SOR ADD L192:11 1 L192:11 EOR
%   L192:11  BOT_COUNT %
% Rung: 1 %
% used for speed calculations %
SOR RHC L192:0 EOR
%   L192:0  BOT_THIS_TIME  "rtc bot belt movement event time" %
% Rung: 2 %
SOR ADD L192:3 1 L192:3 EOR
%   L192:3  BOT_LOOP_COUNT %
% Rung: 3 %
SOR OTU S:5/0 EOR
%   S:5/0  "Overflow Trap" %
% Rung: 4 %
SOR END EOR

LADDER 100 "1 MS STI"    % high speed %
